(* IEC 61131-3 sources: CodesysTest/alpha/export/Pro18_1174_HilscherCard.dev/Plc Logic/Application/Motors/Applied Motion/FB_AppliedMotionStepServoEIPBaseQX.pou/Moving.prop, 1 file *)

(* ---- Get.pm.st ---- *)
(*#-#-#-#-#-#-#-#-#-#---Declaration---#-#-#-#-#-#-#-#-#-#-#-#-#*)

VAR
END_VAR
(*#-#-#-#-#-#-#-#-#-#---Implementation---#-#-#-#-#-#-#-#-#-#-#-#-#*)

Moving := status.moving;
